(*! <Summary>
Fluent interface for full string building and manipulation.
</Summary> *)
INTERFACE IStringBuilder

METHOD Append : IStringBuilder // Returns the builder for fluent chaining.
VAR_INPUT
	Text : STRING(GVL_Param_AUT_Utilities.StringBuilder_MaxStringLength); // Text to append to the current built string
END_VAR
END_METHOD

METHOD AppendWithFormat : IStringBuilder // Returns the builder for fluent chaining.
VAR_INPUT
	Value : ANY;    // Value to format (any primitive type)
	Format : STRING(GVL_Param_AUT_Utilities.StringBuilder_MaxStringLength); // Printf-style format string (e.g. '%05d', '%.2f', '%X')
END_VAR
END_METHOD

METHOD AssignDelimitedSubstringTo : IStringBuilder // Returns the builder for fluent chaining.
VAR_INPUT
    Delimiter : STRING(1); // Single-character delimiter
    SubstringIndex : UDINT; // 1-based index of the token to extract (0 returns empty string)
	Destination : POINTER TO STRING(GVL_Param_AUT_Utilities.StringBuilder_MaxStringLength); // Pointer to the destination string
    DestinationSize : UDINT; // Size in bytes of the destination string
END_VAR
END_METHOD

METHOD AssignTo : IStringBuilder // Returns the builder for fluent chaining.
VAR_INPUT
	Destination : POINTER TO STRING(GVL_Param_AUT_Utilities.StringBuilder_MaxStringLength); // Pointer to the destination string
    DestinationSize : UDINT; // Size in bytes of the destination string
END_VAR
END_METHOD

METHOD InsertAt : IStringBuilder // Returns the builder for fluent chaining.
VAR_INPUT
	Text : STRING(GVL_Param_AUT_Utilities.StringBuilder_MaxStringLength); // Text to insert
	Position : UDINT; // 1-based position at which to insert the text
END_VAR
END_METHOD

METHOD Left : IStringBuilder // Returns the builder for fluent chaining.
VAR_INPUT
	Length : UDINT; // Number of characters to keep from the left
END_VAR
END_METHOD

METHOD Mid : IStringBuilder // Returns the builder for fluent chaining.
VAR_INPUT
	Position : UDINT; // 1-based starting position
	Length : UDINT; // Number of characters to keep
END_VAR
END_METHOD

METHOD PadLeft : IStringBuilder // Returns the builder for fluent chaining.
VAR_INPUT
    PaddingChar : STRING(1); // Single character used for padding
	TotalLength : UDINT; // Desired total length after padding
END_VAR
END_METHOD

METHOD PadRight : IStringBuilder // Returns the builder for fluent chaining.
VAR_INPUT
    PaddingChar : STRING(1); // Single character used for padding
	TotalLength : UDINT; // Desired total length after padding
END_VAR
END_METHOD

METHOD RemoveAt : IStringBuilder // Returns the builder for fluent chaining.
VAR_INPUT
	Position : UDINT; // 1-based position from which to start removing
    Length : UDINT; // Number of characters to remove
END_VAR
END_METHOD

METHOD RemoveDelimitedSubstring : IStringBuilder // Returns the builder for fluent chaining.
VAR_INPUT
    Delimiter : STRING(1); // Single-character delimiter
    SubstringIndex : UDINT; // 1-based index of the token to remove
END_VAR
END_METHOD

METHOD ReplaceAt : IStringBuilder // Returns the builder for fluent chaining.
VAR_INPUT
    Text : STRING(GVL_Param_AUT_Utilities.StringBuilder_MaxStringLength); // Replacement text
	Position : UDINT; // 1-based position of the first character to replace
    Length : UDINT; // Number of characters to replace
END_VAR
END_METHOD

METHOD Reset : ILimitedStringBuilder // Returns the limited builder interface for fluent chaining.
END_METHOD

METHOD Right : IStringBuilder // Returns the builder for fluent chaining.
VAR_INPUT
	Length : UDINT; // Number of characters to keep from the right
END_VAR
END_METHOD

METHOD ToString : STRING(GVL_Param_AUT_Utilities.StringBuilder_MaxStringLength) // The current built string.
END_METHOD

METHOD ToWString : WSTRING(GVL_Param_AUT_Utilities.StringBuilder_MaxStringLength) // The current built string as WSTRING.
END_METHOD

END_INTERFACE

(* stored: Version 1.1.0.1
   Itf IStringBuilder: Id {a96f9cef-4f33-4ae4-9622-b562253d04a0}
   Method Append: Id {5802eef8-4768-447d-ac88-e4a7e9a4f4d4}
   Method AppendWithFormat: Id {df05e3dc-baf8-4636-8c44-47459edd0d1f}
   Method AssignDelimitedSubstringTo: Id {f8790f8f-2557-4c2d-a39d-d6daaf698cf6}
   Method AssignTo: Id {c9769b97-efb5-4d30-8683-906edf176a90}
   Method InsertAt: Id {240a8eb2-830b-47ca-9391-a327b097efb3}
   Method Left: Id {6d0c8a7a-145c-4460-9161-51ed4c634dd3}
   Method Mid: Id {dc588605-d43e-4708-9622-8e4396e24184}
   Method PadLeft: Id {1d9fd8ae-5b0d-4653-9f60-32a24a7b6e77}
   Method PadRight: Id {e629a050-5959-4310-a785-f6d38597d96e}
   Method RemoveAt: Id {ff04897d-a67c-4131-a8d9-c2aed5c52ac3}
   Method RemoveDelimitedSubstring: Id {a4e60b66-0e3c-4e6e-a56f-5cfb7268a908}
   Method ReplaceAt: Id {043e6c07-bfa2-4e4b-8723-2fd1257be72d}
   Method Reset: Id {6597caa0-da9c-4a84-b85b-7d02773d9b7d}
   Method Right: Id {8ab9a4b3-8843-44ac-9824-dcff801059b3}
   Method ToString: Id {acbc2342-d0e7-452e-9b07-7dea4bd95d81}
   Method ToWString: Id {65b50ad9-a317-4856-a5b6-0ed46815bd97} *)
